Staubli VAL3: PointGrey.dtx

public bool bCalibrating
bool bDebug = true
public bool bTaskDetOK
num hCamTable = 1
num nLatchedValue[10]
public num nMaxNumOfObject = 10
public num nNumOfPart = -1
num nObjectID[10]
  [0] = -1
  [1] = -1
  [2] = -1
  [3] = -1
  [4] = -1
  [5] = -1
  [6] = -1
  [7] = -1
  [8] = -1
  [9] = -1
object oTempQueue[10]
  [0]
    num nID = 1
    num nLatchedValue
    trsf trTrsf = {x=32.4, y=22.9, rz=134}
  [1]
    num nID = 1
    num nLatchedValue
    trsf trTrsf = {x=-138.4, y=13.1, rz=115.7}
  [2]
    num nID
    num nLatchedValue
    trsf trTrsf
  [3]
    num nID
    num nLatchedValue
    trsf trTrsf
  [4]
    num nID
    num nLatchedValue
    trsf trTrsf
  [5]
    num nID
    num nLatchedValue
    trsf trTrsf
  [6]
    num nID
    num nLatchedValue
    trsf trTrsf
  [7]
    num nID
    num nLatchedValue
    trsf trTrsf
  [8]
    num nID
    num nLatchedValue
    trsf trTrsf
  [9]
    num nID
    num nLatchedValue
    trsf trTrsf
screen scVision
sio skVision = {link=Socket\PointGrey}
string sDetNum = "DET0"
string sTASK = "detect0"
string strError
trsf trObjectPos[10]
